# EPICS substitutions: ek9000App/Db/EL4024.substitutions
file EL4024.template
{       pattern
        {
                TERMINAL,

        }
        {
        }
}
